INTERFACE I_Resettable

METHOD Reset : BOOL
END_METHOD

END_INTERFACE

(* stored: Version 1.1.0.1, ProductVersion 3.1.4024.12
   Itf I_Resettable: Id {12387b17-1185-4d94-9d20-f45f31d70af6}
   Method Reset: Id {f9ebbe92-edd0-4594-8871-7d5508be33dd} *)
